FUNCTION_BLOCK KinematicControl
VAR
	
	_Master				: MasterAxisControl;
	_Slave				: ARRAY [1.._NumOfSlaves] OF SlaveAxisControl;
	
	_LocalState			: BYTE;
	_i					: BYTE;
	
END_VAR
VAR CONSTANT
	
	_NumOfSlaves		: BYTE := 3;

END_VAR

METHOD CyclicUpdate : BOOL
VAR_INPUT
END_VAR

// Update all axes
_Master.CyclicUpdate();
FOR _i := 1 TO _NumOfSlaves BY 1 DO
	_Slave[_i].CyclicUpdate();
END_FOR

_Slave[1].PreviousAnglePosition 	:= _Master.AnglePosition;
_Slave[1].PreviousLengthOfShaft 	:= _Master.LengthOfShaft;
_Slave[1].PreviousWidthOfShaft		:= _Master.WidthOfShaft;
_Slave[1].PreviousXCoordGlobal		:= _Master.XCoord;
_Slave[1].PreviousYCoordGlobal		:= _Master.YCoord;

IF _NumOfSlaves > 1 THEN
	FOR _i := 2 TO _NumOfSlaves BY 1 DO
		_Slave[_i].PreviousAnglePosition	:= _Slave[_i - 1].AnglePosition;
		_Slave[_i].PreviousLengthOfShaft 	:= _Slave[_i - 1].LengthOfShaft;
		_Slave[_i].PreviousWidthOfShaft		:= _Slave[_i - 1].WidthOfShaft;
		_Slave[_i].PreviousXCoordGlobal		:= _Slave[_i - 1].XCoord;
		_Slave[_i].PreviousYCoordGlobal		:= _Slave[_i - 1].YCoord;
	END_FOR	
END_IF
END_METHOD

END_FUNCTION_BLOCK

(* stored: Version 1.1.0.1, ProductVersion 3.1.4024.12
   POU KinematicControl: Id {de91caef-386b-43ef-9c44-406dad6ca978}, SpecialFunc None
   Method CyclicUpdate: Id {a1c7abaa-811c-40fd-8aa1-380b619fe4b2} *)
